/// SoE commands
TYPE E_SoECommand :
(
	eSoECommand_none := 0,
	eSoECommand_writeIndraDrvPos
);
END_TYPE

(* stored: Version 1.1.0.1, ProductVersion 3.1.4020.12
   DUT E_SoECommand: Id {d63eae55-a98e-4cf7-96d1-59129fcf49c1} *)
